// Mitsubishi GX Works2 project: motionplc   PLC: FX3U/FX3UC

PROGRAM MAIN
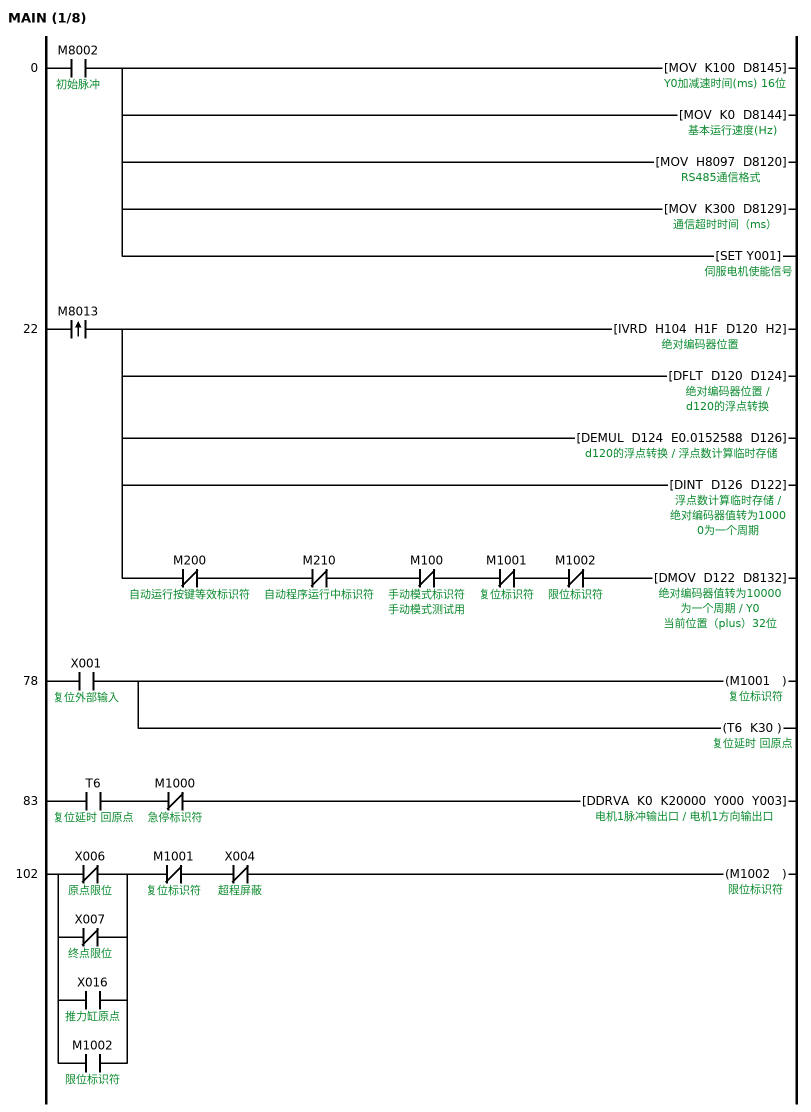
0     LD      M8002  ; 初始脉冲
      MOV     K100 D8145  ; Y0加减速时间(ms) 16位
      MOV     K0 D8144  ; 基本运行速度(Hz)
      MOV     H8097 D8120  ; RS485通信格式
      MOV     K300 D8129  ; 通信超时时间（ms）
      SET     Y001  ; 伺服电机使能信号
22    LDP     M8013
      IVRD    H104 H1F D120 H2  ; 绝对编码器位置
      DFLT    D120 D124  ; d120的浮点转换
      DEMUL   D124 E0.0152588 D126  ; 浮点数计算临时存储
      DINT    D126 D122  ; 绝对编码器值转为10000为一个周期
      ANI     M200  ; 自动运行按键等效标识符
      ANI     M210  ; 自动程序运行中标识符
      ANI     M100  ; 手动模式标识符 手动模式测试用
      ANI     M1001  ; 复位标识符
      ANI     M1002  ; 限位标识符
      DMOV    D122 D8132  ; Y0 当前位置（plus）32位
78    LD      X001  ; 复位外部输入
      OUT     M1001  ; 复位标识符
      OUT     T6 K30  ; 复位延时 回原点
83    LD      T6  ; 复位延时 回原点
      ANI     M1000  ; 急停标识符
      DDRVA   K0 K20000 Y000 Y003  ; 电机1脉冲输出口 / 电机1方向输出口
102   LDI     X006  ; 原点限位
      ORI     X007  ; 终点限位
      OR      X016  ; 推力缸原点
      OR      M1002  ; 限位标识符
      ANI     M1001  ; 复位标识符
      ANI     X004  ; 超程屏蔽
      OUT     M1002  ; 限位标识符
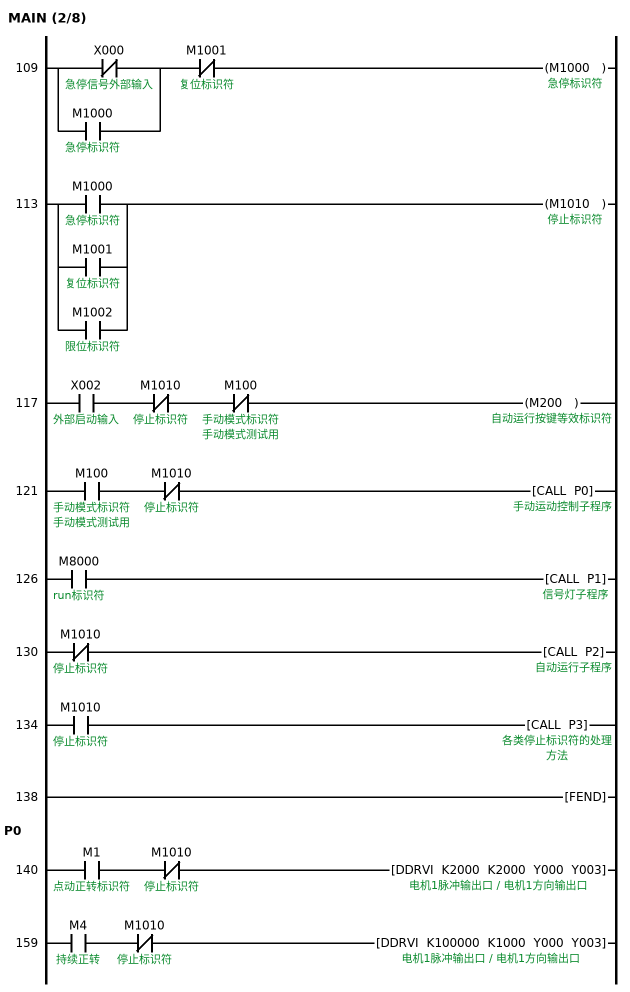
109   LDI     X000  ; 急停信号外部输入
      OR      M1000  ; 急停标识符
      ANI     M1001  ; 复位标识符
      OUT     M1000  ; 急停标识符
113   LD      M1000  ; 急停标识符
      OR      M1001  ; 复位标识符
      OR      M1002  ; 限位标识符
      OUT     M1010  ; 停止标识符
117   LD      X002  ; 外部启动输入
      ANI     M1010  ; 停止标识符
      ANI     M100  ; 手动模式标识符 手动模式测试用
      OUT     M200  ; 自动运行按键等效标识符
121   LD      M100  ; 手动模式标识符 手动模式测试用
      ANI     M1010  ; 停止标识符
      CALL    P0  ; 手动运动控制子程序
126   LD      M8000  ; run标识符
      CALL    P1  ; 信号灯子程序
130   LDI     M1010  ; 停止标识符
      CALL    P2  ; 自动运行子程序
134   LD      M1010  ; 停止标识符
      CALL    P3  ; 各类停止标识符的处理方法
138   FEND
      P0
140   LD      M1  ; 点动正转标识符
      ANI     M1010  ; 停止标识符
      DDRVI   K2000 K2000 Y000 Y003
159   LD      M4  ; 持续正转
      ANI     M1010  ; 停止标识符
      DDRVI   K100000 K1000 Y000 Y003
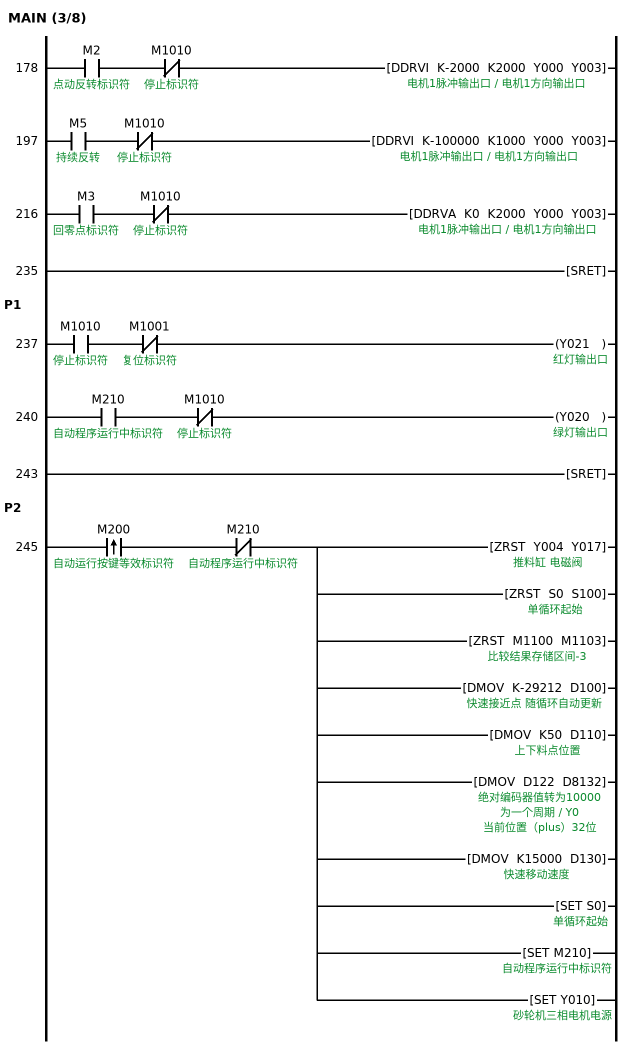
178   LD      M2  ; 点动反转标识符
      ANI     M1010  ; 停止标识符
      DDRVI   K-2000 K2000 Y000 Y003
197   LD      M5  ; 持续反转
      ANI     M1010  ; 停止标识符
      DDRVI   K-100000 K1000 Y000 Y003
216   LD      M3  ; 回零点标识符
      ANI     M1010  ; 停止标识符
      DDRVA   K0 K2000 Y000 Y003
235   SRET
      P1
237   LD      M1010  ; 停止标识符
      ANI     M1001  ; 复位标识符
      OUT     Y021  ; 红灯输出口
240   LD      M210  ; 自动程序运行中标识符
      ANI     M1010  ; 停止标识符
      OUT     Y020  ; 绿灯输出口
243   SRET
      P2
245   LDP     M200  ; 自动运行按键等效标识符
      ANI     M210  ; 自动程序运行中标识符
      ZRST    Y004 Y017  ; 推料缸 电磁阀
      ZRST    S0 S100  ; 单循环起始
      ZRST    M1100 M1103  ; 比较结果存储区间-3
      DMOV    K-29212 D100  ; 快速接近点 随循环自动更新
      DMOV    K50 D110  ; 上下料点位置
      DMOV    D122 D8132
      DMOV    K15000 D130  ; 快速移动速度
      SET     S0  ; 单循环起始
      SET     M210  ; 自动程序运行中标识符
      SET     Y010  ; 砂轮机三相电机电源
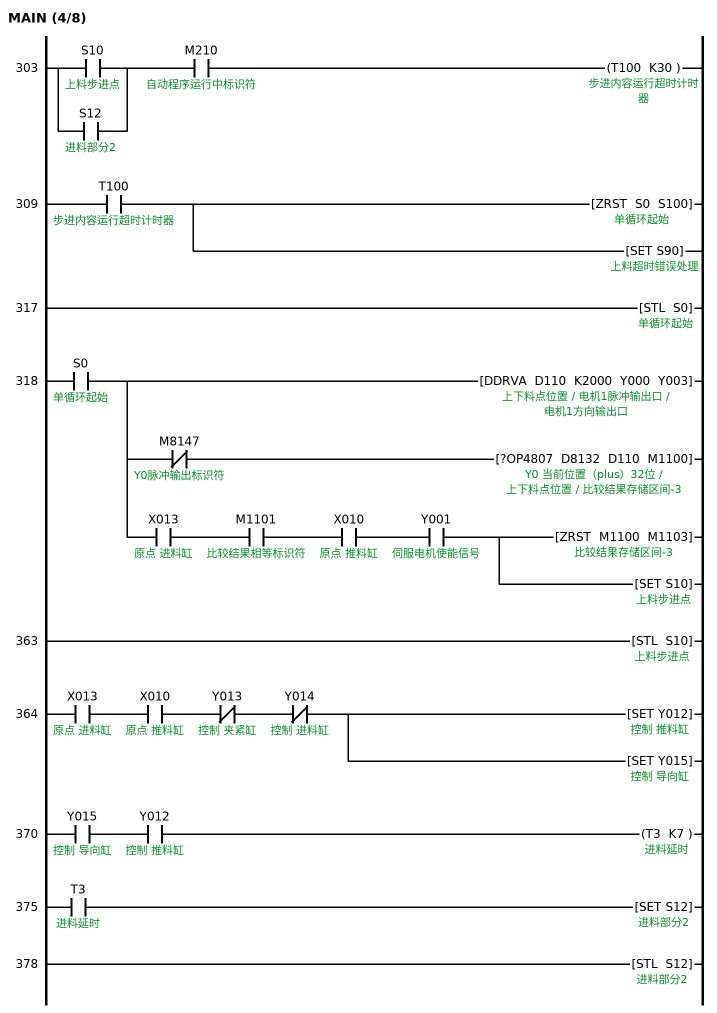
303   LD      S10  ; 上料步进点
      OR      S12  ; 进料部分2
      AND     M210  ; 自动程序运行中标识符
      OUT     T100 K30  ; 步进内容运行超时计时器
309   LD      T100  ; 步进内容运行超时计时器
      ZRST    S0 S100
      SET     S90  ; 上料超时错误处理
317   STL     S0
318   LD      S0  ; 单循环起始
      DDRVA   D110 K2000 Y000 Y003
      MPS
      ANI     M8147  ; Y0脉冲输出标识符
      ?OP4807 D8132 D110 M1100
      MPP
      AND     X013  ; 原点 进料缸
      AND     M1101  ; 比较结果相等标识符
      AND     X010  ; 原点 推料缸
      AND     Y001  ; 伺服电机使能信号
      ZRST    M1100 M1103
      SET     S10  ; 上料步进点
363   STL     S10
364   LD      X013  ; 原点 进料缸
      AND     X010  ; 原点 推料缸
      ANI     Y013  ; 控制 夹紧缸
      ANI     Y014  ; 控制 进料缸
      SET     Y012  ; 控制 推料缸
      SET     Y015  ; 控制 导向缸
370   LD      Y015  ; 控制 导向缸
      AND     Y012  ; 控制 推料缸
      OUT     T3 K7  ; 进料延时
375   LD      T3  ; 进料延时
      SET     S12  ; 进料部分2
378   STL     S12
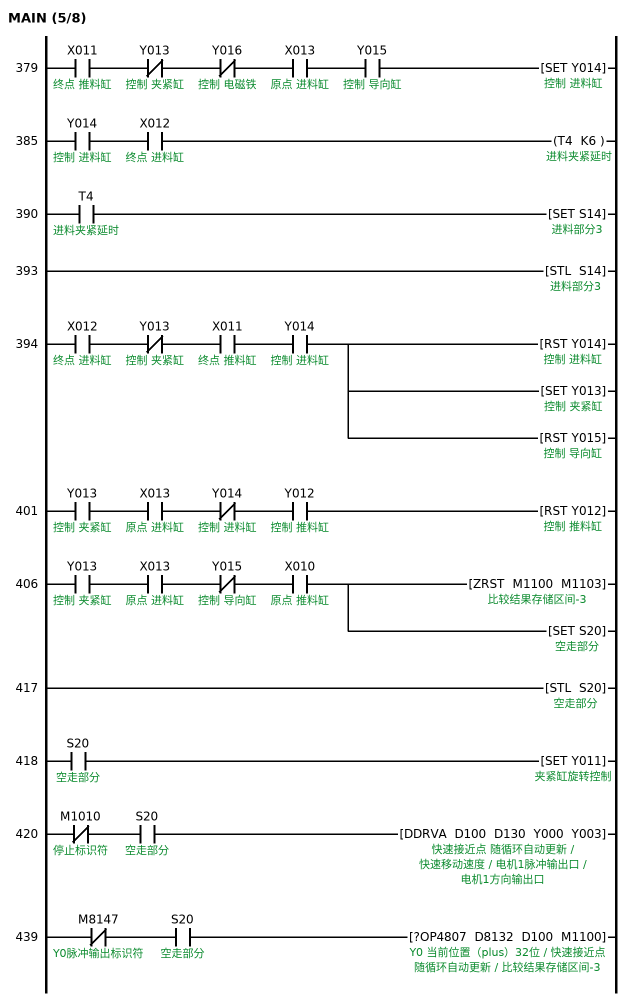
379   LD      X011  ; 终点 推料缸
      ANI     Y013  ; 控制 夹紧缸
      ANI     Y016  ; 控制 电磁铁
      AND     X013  ; 原点 进料缸
      AND     Y015  ; 控制 导向缸
      SET     Y014  ; 控制 进料缸
385   LD      Y014  ; 控制 进料缸
      AND     X012  ; 终点 进料缸
      OUT     T4 K6  ; 进料夹紧延时
390   LD      T4  ; 进料夹紧延时
      SET     S14  ; 进料部分3
393   STL     S14
394   LD      X012  ; 终点 进料缸
      ANI     Y013  ; 控制 夹紧缸
      AND     X011  ; 终点 推料缸
      AND     Y014  ; 控制 进料缸
      RST     Y014  ; 控制 进料缸
      SET     Y013  ; 控制 夹紧缸
      RST     Y015  ; 控制 导向缸
401   LD      Y013  ; 控制 夹紧缸
      AND     X013  ; 原点 进料缸
      ANI     Y014  ; 控制 进料缸
      AND     Y012  ; 控制 推料缸
      RST     Y012  ; 控制 推料缸
406   LD      Y013  ; 控制 夹紧缸
      AND     X013  ; 原点 进料缸
      ANI     Y015  ; 控制 导向缸
      AND     X010  ; 原点 推料缸
      ZRST    M1100 M1103
      SET     S20  ; 空走部分
417   STL     S20
418   LD      S20  ; 空走部分
      SET     Y011  ; 夹紧缸旋转控制
420   LDI     M1010  ; 停止标识符
      AND     S20  ; 空走部分
      DDRVA   D100 D130 Y000 Y003
439   LDI     M8147  ; Y0脉冲输出标识符
      AND     S20  ; 空走部分
      ?OP4807 D8132 D100 M1100
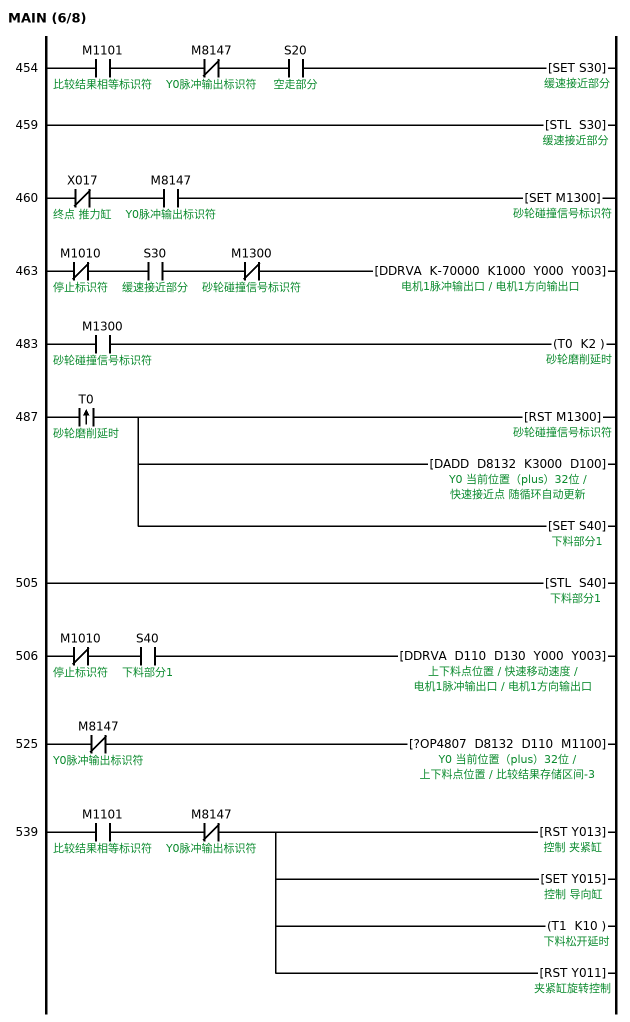
454   LD      M1101  ; 比较结果相等标识符
      ANI     M8147  ; Y0脉冲输出标识符
      AND     S20  ; 空走部分
      SET     S30  ; 缓速接近部分
459   STL     S30
460   LDI     X017  ; 终点 推力缸
      AND     M8147  ; Y0脉冲输出标识符
      SET     M1300  ; 砂轮碰撞信号标识符
463   LDI     M1010  ; 停止标识符
      AND     S30  ; 缓速接近部分
      ANI     M1300  ; 砂轮碰撞信号标识符
      DDRVA   K-70000 K1000 Y000 Y003
483   LD      M1300  ; 砂轮碰撞信号标识符
      OUT     T0 K2  ; 砂轮磨削延时
487   LDP     T0  ; 砂轮磨削延时
      RST     M1300  ; 砂轮碰撞信号标识符
      DADD    D8132 K3000 D100
      SET     S40  ; 下料部分1
505   STL     S40
506   LDI     M1010  ; 停止标识符
      AND     S40  ; 下料部分1
      DDRVA   D110 D130 Y000 Y003
525   LDI     M8147  ; Y0脉冲输出标识符
      ?OP4807 D8132 D110 M1100
539   LD      M1101  ; 比较结果相等标识符
      ANI     M8147  ; Y0脉冲输出标识符
      RST     Y013  ; 控制 夹紧缸
      SET     Y015  ; 控制 导向缸
      OUT     T1 K10  ; 下料松开延时
      RST     Y011  ; 夹紧缸旋转控制
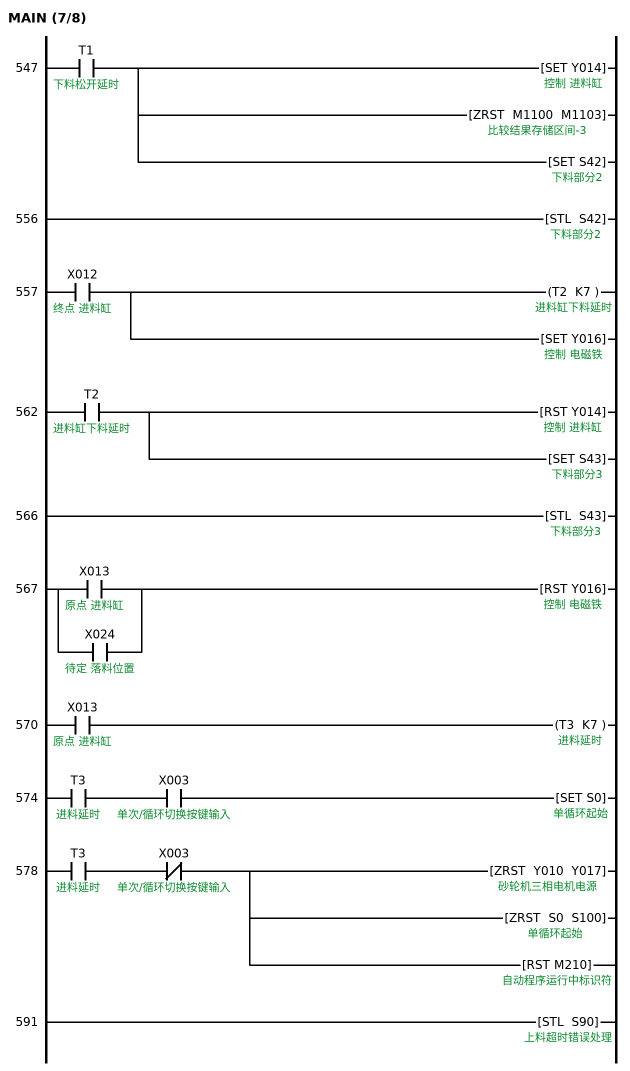
547   LD      T1  ; 下料松开延时
      SET     Y014  ; 控制 进料缸
      ZRST    M1100 M1103
      SET     S42  ; 下料部分2
556   STL     S42
557   LD      X012  ; 终点 进料缸
      OUT     T2 K7  ; 进料缸下料延时
      SET     Y016  ; 控制 电磁铁
562   LD      T2  ; 进料缸下料延时
      RST     Y014  ; 控制 进料缸
      SET     S43  ; 下料部分3
566   STL     S43
567   LD      X013  ; 原点 进料缸
      OR      X024  ; 待定 落料位置
      RST     Y016  ; 控制 电磁铁
570   LD      X013  ; 原点 进料缸
      OUT     T3 K7  ; 进料延时
574   LD      T3  ; 进料延时
      AND     X003  ; 单次/循环切换按键输入
      SET     S0  ; 单循环起始
578   LD      T3  ; 进料延时
      ANI     X003  ; 单次/循环切换按键输入
      ZRST    Y010 Y017
      ZRST    S0 S100
      RST     M210  ; 自动程序运行中标识符
591   STL     S90
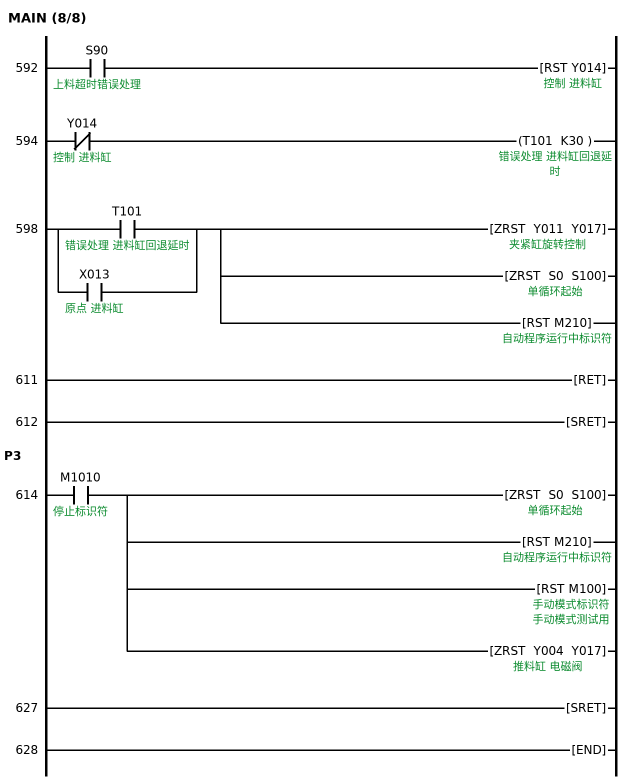
592   LD      S90  ; 上料超时错误处理
      RST     Y014  ; 控制 进料缸
594   LDI     Y014  ; 控制 进料缸
      OUT     T101 K30  ; 错误处理 进料缸回退延时
598   LD      T101  ; 错误处理 进料缸回退延时
      OR      X013  ; 原点 进料缸
      ZRST    Y011 Y017
      ZRST    S0 S100
      RST     M210  ; 自动程序运行中标识符
611   RET
612   SRET
      P3
614   LD      M1010  ; 停止标识符
      ZRST    S0 S100
      RST     M210  ; 自动程序运行中标识符
      RST     M100  ; 手动模式标识符 手动模式测试用
      ZRST    Y004 Y017
627   SRET
628   END
END_PROGRAM

// device comments not shown above
Y005  ; 进料缸
Y006  ; 夹紧缸
Y007  ; 导向缸电磁阀
D200  ; 临时存储位置判定数据
M201  ; 自动程序 运行初始化
M203  ; 上料部分
M205  ; 空走部分
M207  ; 慢速接近砂轮部分
M1003  ; 自动程序步进点运行超时标识符
M1400  ; 位置比较结果
M1401  ; 比较结果相等标识符
M1500  ; 测试用 屏蔽停止标识符
X005  ; 超程屏蔽
X020  ; 气缸落料位置
X022  ; 循环标识符
S41  ; 下料松开部分2
T10  ; 步进点1 超时计时器
T102  ; 上料步骤1超时
T104  ; 上料步骤2超时 无料进料缸超位置
T106  ; 上料结束步骤超时计时器
T110  ; 上料步骤1超时
